Fanuc KAREL source: kd00070.KL

-- PROVISIONAL review KL for V770-1; original PC SHA256 fcb3b49c2f15cb479c3d7db0204573e5545e60a7d52980928eb561333073a094
-- Incomplete behavior may be omitted. Consult companion uncertainty JSON. Do not deploy.
PROGRAM KD00070
%NOLOCKGROUP
VAR
  I : INTEGER
  J : INTEGER
  B : BOOLEAN
  R : REAL
  S : STRING[80]
BEGIN
  -- UNRESOLVED_PC offsets 5-18; opcodes 9D,81,18,9D,1B,9D,12,9C,13,04
  -- UNRESOLVED_PC offsets 23-27; opcodes 7F
END KD00070
